SYSTEM TESTBED_MVCL (* Testbed Model/View/Control with Local Coupling *)
  (* Standard: 61499 ITA; Classification: Testbed *)
  (* Version 0.3, 2004-11-09, JHC, Rockwell Automation, Changed LOADL to LOADLE in CHAIN_MDL. *)
  (* Version 0.2, 2004-10-28, JHC, Rockwell Automation, Changed RING_FEED to CNVG_MDLL. *)
  (* Version 0.1, 2004-10-25, JHC, Rockwell Automation, Updated for new Load/Unload model. *)
  (* Version 0.0, 2004-09-22, JHC, Rockwell Automation *)
  DEVICE CONTROL : FRAME_DEVICE
    RESOURCE SORT : EMB_RES
      FBS
        SORT_PEG_SENSE : SUBL_2;
        RING_FEED_SENSE : SUBL_1;
        CTL : SORT_CTL;
        SORT_ACT : PUBL_1;
        LOST : E_PERMIT; (* RING_LOST event trigger *)
        RING_LOST : PUBL_0;
      END_FBS
      EVENT_CONNECTIONS
        START.COLD TO SORT_PEG_SENSE.INIT;
        SORT_PEG_SENSE.INITO TO RING_FEED_SENSE.INIT;
        RING_FEED_SENSE.INITO TO SORT_ACT.INIT;
        SORT_PEG_SENSE.IND TO CTL.REQ;
        CTL.CNF TO SORT_ACT.REQ;
        CTL.CNF TO LOST.EI;
        SORT_ACT.INITO TO RING_LOST.INIT;
        LOST.EO TO RING_LOST.REQ;
      END_CONNECTIONS
      DATA_CONNECTIONS
        RING_FEED_SENSE.RD_1 TO CTL.RING_PRESENT;
        CTL.SORT_SOLENOID TO SORT_ACT.SD_1;
        SORT_PEG_SENSE.RD_1 TO CTL.SORT_AREA_DETECT;
        SORT_PEG_SENSE.RD_2 TO CTL.METAL_PEG_DETECT;
        CTL.RING_LOST TO LOST.PERMIT;
      END_CONNECTIONS
    END_RESOURCE
    RESOURCE FEED : EMB_RES
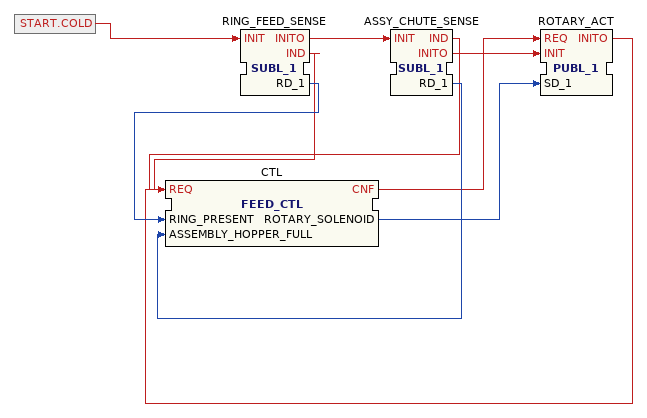
      FBS
        RING_FEED_SENSE : SUBL_1;
        ASSY_CHUTE_SENSE : SUBL_1;
        CTL : FEED_CTL;
        ROTARY_ACT : PUBL_1;
      END_FBS
      EVENT_CONNECTIONS
        START.COLD TO RING_FEED_SENSE.INIT;
        RING_FEED_SENSE.INITO TO ASSY_CHUTE_SENSE.INIT;
        ROTARY_ACT.INITO TO CTL.REQ;
        RING_FEED_SENSE.IND TO CTL.REQ;
        ASSY_CHUTE_SENSE.IND TO CTL.REQ;
        CTL.CNF TO ROTARY_ACT.REQ;
        ASSY_CHUTE_SENSE.INITO TO ROTARY_ACT.INIT;
      END_CONNECTIONS
      DATA_CONNECTIONS
        RING_FEED_SENSE.RD_1 TO CTL.RING_PRESENT;
        ASSY_CHUTE_SENSE.RD_1 TO CTL.ASSEMBLY_HOPPER_FULL;
        CTL.ROTARY_SOLENOID TO ROTARY_ACT.SD_1;
      END_CONNECTIONS
    END_RESOURCE
    RESOURCE INSPECT : EMB_RES
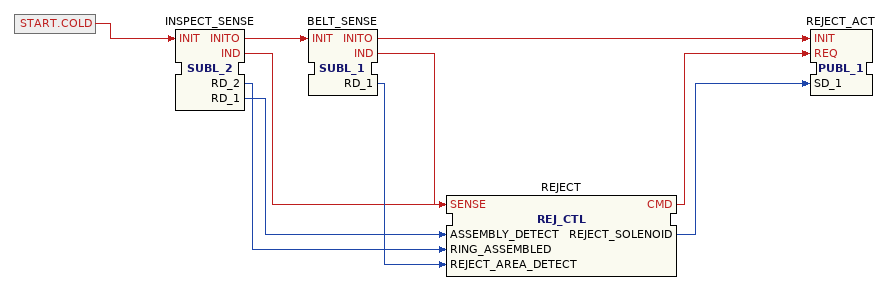
      FBS
        INSPECT_SENSE : SUBL_2;
        BELT_SENSE : SUBL_1;
        REJECT_ACT : PUBL_1;
        REJECT : REJ_CTL;
      END_FBS
      EVENT_CONNECTIONS
        START.COLD TO INSPECT_SENSE.INIT;
        INSPECT_SENSE.INITO TO BELT_SENSE.INIT;
        BELT_SENSE.INITO TO REJECT_ACT.INIT;
        INSPECT_SENSE.IND TO REJECT.SENSE;
        BELT_SENSE.IND TO REJECT.SENSE;
        REJECT.CMD TO REJECT_ACT.REQ;
      END_CONNECTIONS
      DATA_CONNECTIONS
        REJECT.REJECT_SOLENOID TO REJECT_ACT.SD_1;
        INSPECT_SENSE.RD_2 TO REJECT.RING_ASSEMBLED;
        INSPECT_SENSE.RD_1 TO REJECT.ASSEMBLY_DETECT;
        BELT_SENSE.RD_1 TO REJECT.REJECT_AREA_DETECT;
      END_CONNECTIONS
    END_RESOURCE
    RESOURCE CHAIN_SENSORS : PANEL_RESOURCE
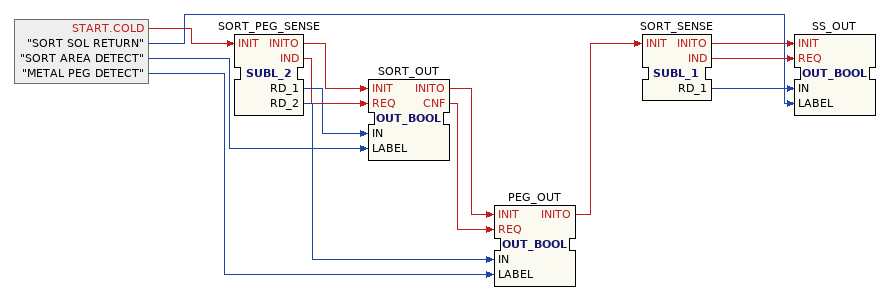
      FBS
        SORT_SENSE : SUBL_1;
        SS_OUT : OUT_BOOL;
        SORT_PEG_SENSE : SUBL_2;
        PEG_OUT : OUT_BOOL;
        SORT_OUT : OUT_BOOL;
      END_FBS
      EVENT_CONNECTIONS
        SORT_PEG_SENSE.INITO TO SORT_OUT.INIT;
        SORT_PEG_SENSE.IND TO SORT_OUT.REQ;
        SORT_OUT.INITO TO PEG_OUT.INIT;
        SORT_OUT.CNF TO PEG_OUT.REQ;
        START.COLD TO SORT_PEG_SENSE.INIT;
        PEG_OUT.INITO TO SORT_SENSE.INIT;
        SORT_SENSE.INITO TO SS_OUT.INIT;
        SORT_SENSE.IND TO SS_OUT.REQ;
      END_CONNECTIONS
      DATA_CONNECTIONS
        SORT_SENSE.RD_1 TO SS_OUT.IN;
        SORT_PEG_SENSE.RD_1 TO SORT_OUT.IN;
        SORT_PEG_SENSE.RD_2 TO PEG_OUT.IN;
        "SORT SOL RETURN" TO SS_OUT.LABEL;
        "SORT AREA DETECT" TO SORT_OUT.LABEL;
        "METAL PEG DETECT" TO PEG_OUT.LABEL;
      END_CONNECTIONS
    END_RESOURCE
    RESOURCE CHAIN_ACTUATORS : PANEL_RESOURCE
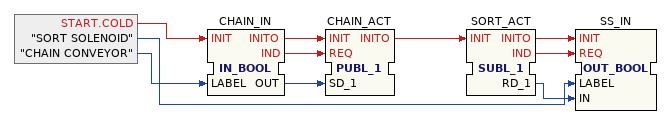
      FBS
        CHAIN_IN : IN_BOOL;
        CHAIN_ACT : PUBL_1;
        SS_IN : OUT_BOOL;
        SORT_ACT : SUBL_1;
      END_FBS
      EVENT_CONNECTIONS
        SORT_ACT.INITO TO SS_IN.INIT;
        SORT_ACT.IND TO SS_IN.REQ;
        START.COLD TO CHAIN_IN.INIT;
        CHAIN_IN.INITO TO CHAIN_ACT.INIT;
        CHAIN_ACT.INITO TO SORT_ACT.INIT;
        CHAIN_IN.IND TO CHAIN_ACT.REQ;
      END_CONNECTIONS
      DATA_CONNECTIONS
        "SORT SOLENOID" TO SS_IN.LABEL;
        "CHAIN CONVEYOR" TO CHAIN_IN.LABEL;
        SORT_ACT.RD_1 TO SS_IN.IN;
        CHAIN_IN.OUT TO CHAIN_ACT.SD_1;
      END_CONNECTIONS
    END_RESOURCE
    RESOURCE CHUTE_SENSORS : PANEL_RESOURCE
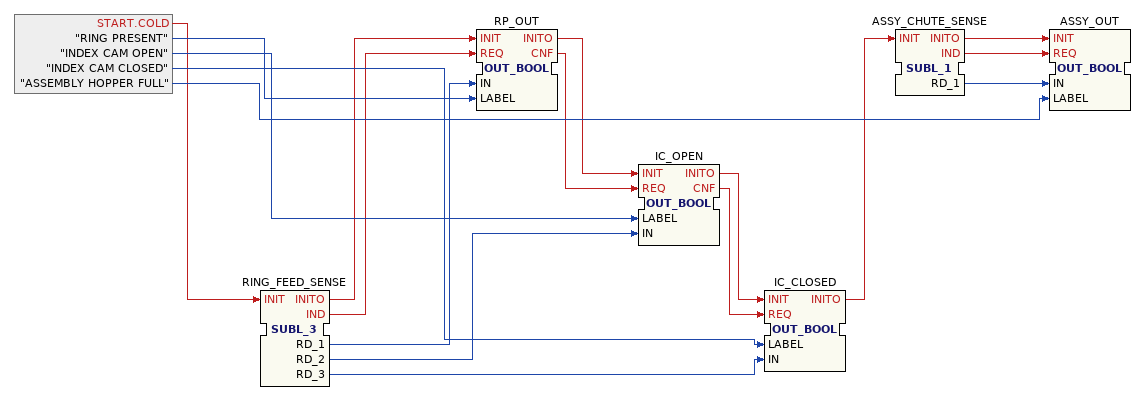
      FBS
        RING_FEED_SENSE : SUBL_3;
        RP_OUT : OUT_BOOL;
        IC_OPEN : OUT_BOOL;
        IC_CLOSED : OUT_BOOL;
        ASSY_CHUTE_SENSE : SUBL_1;
        ASSY_OUT : OUT_BOOL;
      END_FBS
      EVENT_CONNECTIONS
        START.COLD TO RING_FEED_SENSE.INIT;
        RING_FEED_SENSE.INITO TO RP_OUT.INIT;
        IC_OPEN.INITO TO IC_CLOSED.INIT;
        IC_CLOSED.INITO TO ASSY_CHUTE_SENSE.INIT;
        ASSY_CHUTE_SENSE.INITO TO ASSY_OUT.INIT;
        RING_FEED_SENSE.IND TO RP_OUT.REQ;
        IC_OPEN.CNF TO IC_CLOSED.REQ;
        ASSY_CHUTE_SENSE.IND TO ASSY_OUT.REQ;
        RP_OUT.INITO TO IC_OPEN.INIT;
        RP_OUT.CNF TO IC_OPEN.REQ;
      END_CONNECTIONS
      DATA_CONNECTIONS
        RING_FEED_SENSE.RD_1 TO RP_OUT.IN;
        "RING PRESENT" TO RP_OUT.LABEL;
        "INDEX CAM OPEN" TO IC_OPEN.LABEL;
        "INDEX CAM CLOSED" TO IC_CLOSED.LABEL;
        ASSY_CHUTE_SENSE.RD_1 TO ASSY_OUT.IN;
        "ASSEMBLY HOPPER FULL" TO ASSY_OUT.LABEL;
        RING_FEED_SENSE.RD_2 TO IC_OPEN.IN;
        RING_FEED_SENSE.RD_3 TO IC_CLOSED.IN;
      END_CONNECTIONS
    END_RESOURCE
    RESOURCE CHUTE_ACTUATORS : PANEL_RESOURCE
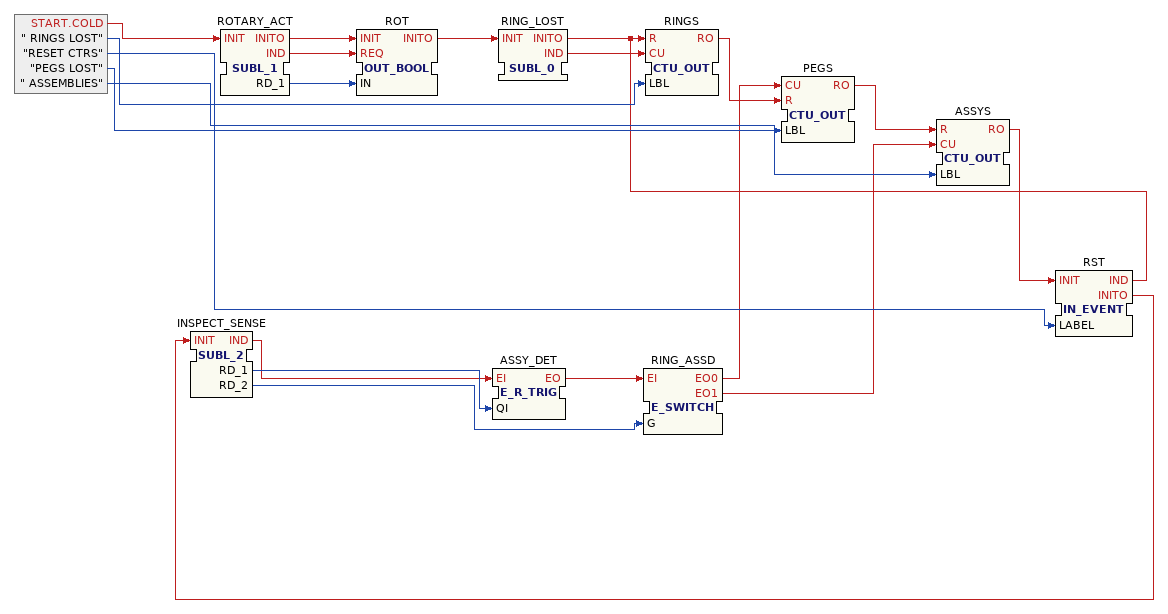
      FBS
        ROT : OUT_BOOL;
        ROTARY_ACT : SUBL_1;
        RING_LOST : SUBL_0;
        RINGS : CTU_OUT;
        RST : IN_EVENT;
        PEGS : CTU_OUT;
        ASSYS : CTU_OUT;
        ASSY_DET : E_R_TRIG; (* QI = ASSEMBLY_DETECT *)
        RING_ASSD : E_SWITCH; (* G = RING_ASSEMBLED *)
        INSPECT_SENSE : SUBL_2;
      END_FBS
      EVENT_CONNECTIONS
        START.COLD TO ROTARY_ACT.INIT;
        ROTARY_ACT.INITO TO ROT.INIT;
        ROTARY_ACT.IND TO ROT.REQ;
        ROT.INITO TO RING_LOST.INIT;
        RING_LOST.INITO TO RINGS.R;
        RING_LOST.IND TO RINGS.CU;
        RST.IND TO RINGS.R;
        ASSYS.RO TO RST.INIT;
        ASSY_DET.EO TO RING_ASSD.EI;
        INSPECT_SENSE.IND TO ASSY_DET.EI;
        RING_ASSD.EO0 TO PEGS.CU;
        RINGS.RO TO PEGS.R;
        PEGS.RO TO ASSYS.R;
        RING_ASSD.EO1 TO ASSYS.CU;
        RST.INITO TO INSPECT_SENSE.INIT;
      END_CONNECTIONS
      DATA_CONNECTIONS
        " RINGS LOST" TO RINGS.LBL;
        "RESET CTRS" TO RST.LABEL;
        "PEGS LOST" TO PEGS.LBL;
        " ASSEMBLIES" TO ASSYS.LBL;
        INSPECT_SENSE.RD_1 TO ASSY_DET.QI;
        INSPECT_SENSE.RD_2 TO RING_ASSD.G;
        ROTARY_ACT.RD_1 TO ROT.IN;
      END_CONNECTIONS
    END_RESOURCE
    RESOURCE BELT_SENSORS : PANEL_RESOURCE
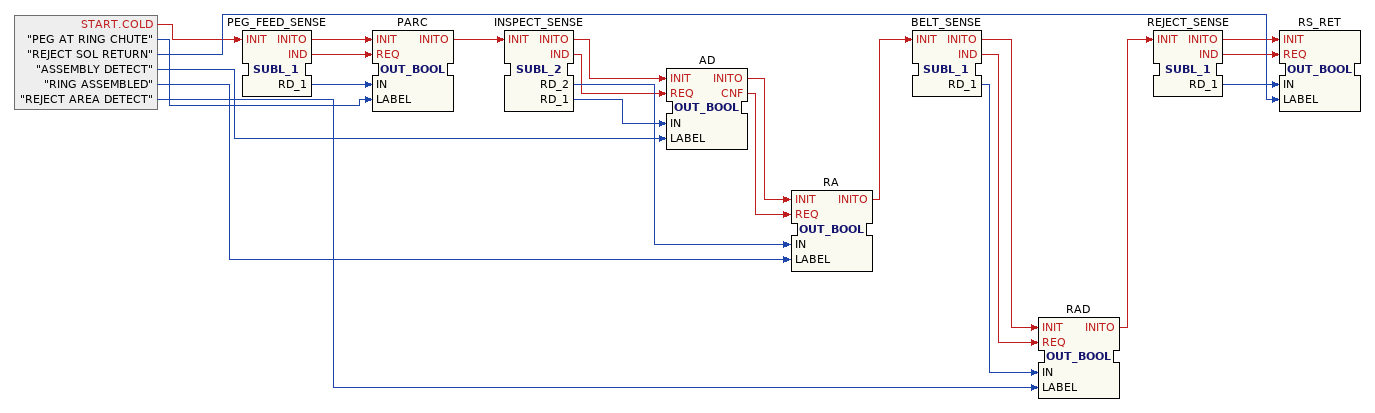
      FBS
        PEG_FEED_SENSE : SUBL_1;
        PARC : OUT_BOOL;
        INSPECT_SENSE : SUBL_2;
        AD : OUT_BOOL;
        RA : OUT_BOOL;
        BELT_SENSE : SUBL_1;
        RAD : OUT_BOOL;
        REJECT_SENSE : SUBL_1;
        RS_RET : OUT_BOOL;
      END_FBS
      EVENT_CONNECTIONS
        START.COLD TO PEG_FEED_SENSE.INIT;
        PEG_FEED_SENSE.INITO TO PARC.INIT;
        PARC.INITO TO INSPECT_SENSE.INIT;
        INSPECT_SENSE.INITO TO AD.INIT;
        AD.INITO TO RA.INIT;
        RA.INITO TO BELT_SENSE.INIT;
        BELT_SENSE.INITO TO RAD.INIT;
        RAD.INITO TO REJECT_SENSE.INIT;
        REJECT_SENSE.INITO TO RS_RET.INIT;
        PEG_FEED_SENSE.IND TO PARC.REQ;
        INSPECT_SENSE.IND TO AD.REQ;
        AD.CNF TO RA.REQ;
        BELT_SENSE.IND TO RAD.REQ;
        REJECT_SENSE.IND TO RS_RET.REQ;
      END_CONNECTIONS
      DATA_CONNECTIONS
        PEG_FEED_SENSE.RD_1 TO PARC.IN;
        "PEG AT RING CHUTE" TO PARC.LABEL;
        REJECT_SENSE.RD_1 TO RS_RET.IN;
        "REJECT SOL RETURN" TO RS_RET.LABEL;
        INSPECT_SENSE.RD_2 TO RA.IN;
        INSPECT_SENSE.RD_1 TO AD.IN;
        "ASSEMBLY DETECT" TO AD.LABEL;
        "RING ASSEMBLED" TO RA.LABEL;
        BELT_SENSE.RD_1 TO RAD.IN;
        "REJECT AREA DETECT" TO RAD.LABEL;
      END_CONNECTIONS
    END_RESOURCE
    RESOURCE BELT_ACTUATORS : PANEL_RESOURCE
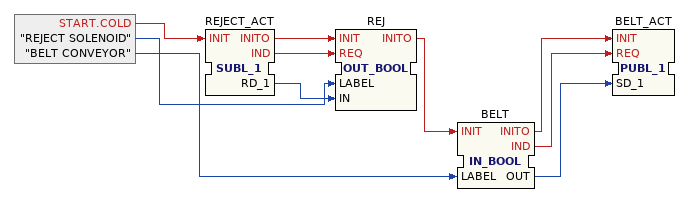
      FBS
        REJ : OUT_BOOL;
        REJECT_ACT : SUBL_1;
        BELT : IN_BOOL;
        BELT_ACT : PUBL_1;
      END_FBS
      EVENT_CONNECTIONS
        BELT.INITO TO BELT_ACT.INIT;
        BELT.IND TO BELT_ACT.REQ;
        START.COLD TO REJECT_ACT.INIT;
        REJECT_ACT.INITO TO REJ.INIT;
        REJECT_ACT.IND TO REJ.REQ;
        REJ.INITO TO BELT.INIT;
      END_CONNECTIONS
      DATA_CONNECTIONS
        "REJECT SOLENOID" TO REJ.LABEL;
        BELT.OUT TO BELT_ACT.SD_1;
        "BELT CONVEYOR" TO BELT.LABEL;
        REJECT_ACT.RD_1 TO REJ.IN;
      END_CONNECTIONS
    END_RESOURCE
  END_DEVICE
  DEVICE MODEL : FRAME_DEVICE
    RESOURCE CLOCK : EMB_RES
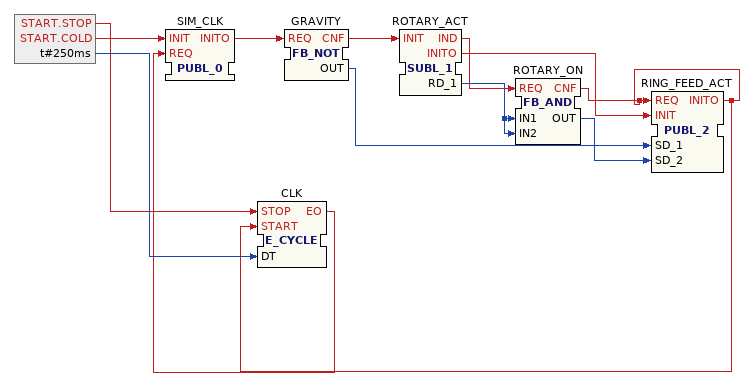
      FBS
        CLK : E_CYCLE;
        SIM_CLK : PUBL_0;
        GRAVITY : FB_NOT;
        ROTARY_ACT : SUBL_1;
        ROTARY_ON : FB_AND;
        RING_FEED_ACT : PUBL_2;
      END_FBS
      EVENT_CONNECTIONS
        START.STOP TO CLK.STOP;
        START.COLD TO SIM_CLK.INIT;
        CLK.EO TO SIM_CLK.REQ;
        SIM_CLK.INITO TO GRAVITY.REQ;
        GRAVITY.CNF TO ROTARY_ACT.INIT;
        ROTARY_ACT.IND TO ROTARY_ON.REQ;
        ROTARY_ON.CNF TO RING_FEED_ACT.REQ;
        ROTARY_ACT.INITO TO RING_FEED_ACT.INIT;
        RING_FEED_ACT.INITO TO RING_FEED_ACT.REQ;
        RING_FEED_ACT.INITO TO CLK.START;
      END_CONNECTIONS
      DATA_CONNECTIONS
        t#250ms TO CLK.DT;
        GRAVITY.OUT TO RING_FEED_ACT.SD_1;
        ROTARY_ACT.RD_1 TO ROTARY_ON.IN1;
        ROTARY_ACT.RD_1 TO ROTARY_ON.IN2;
        ROTARY_ON.OUT TO RING_FEED_ACT.SD_2;
      END_CONNECTIONS
    END_RESOURCE
    RESOURCE CHAIN_MDL : EMB_RES
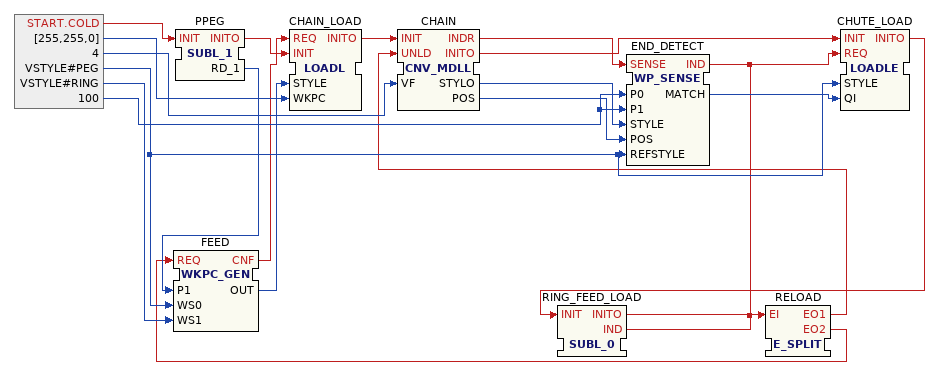
      FBS
        PPEG : SUBL_1;
        FEED : WKPC_GEN;
        CHAIN : CNV_MDLL;
        RING_FEED_LOAD : SUBL_0;
        END_DETECT : WP_SENSE;
        CHAIN_LOAD : LOADL;
        RELOAD : E_SPLIT;
        CHUTE_LOAD : LOADLE;
      END_FBS
      EVENT_CONNECTIONS
        FEED.CNF TO CHAIN_LOAD.REQ;
        START.COLD TO PPEG.INIT;
        PPEG.INITO TO CHAIN_LOAD.INIT;
        CHAIN_LOAD.INITO TO CHAIN.INIT;
        RELOAD.EO1 TO CHAIN.UNLD;
        RELOAD.EO2 TO FEED.REQ;
        RING_FEED_LOAD.INITO TO RELOAD.EI;
        RING_FEED_LOAD.IND TO RELOAD.EI;
        CHAIN.INDR TO END_DETECT.SENSE;
        CHAIN.INITO TO CHUTE_LOAD.INIT;
        CHUTE_LOAD.INITO TO RING_FEED_LOAD.INIT;
        END_DETECT.IND TO CHUTE_LOAD.REQ;
        END_DETECT.IND TO RELOAD.EI;
      END_CONNECTIONS
      DATA_CONNECTIONS
        FEED.OUT TO CHAIN_LOAD.STYLE;
        [255,255,0] TO CHAIN_LOAD.WKPC;
        4 TO CHAIN.VF; (* 16% per sec =100% per 6.25 sec *)
        PPEG.RD_1 TO FEED.P1;
        VSTYLE#PEG TO FEED.WS0;
        VSTYLE#RING TO FEED.WS1;
        100 TO END_DETECT.P0;
        100 TO END_DETECT.P1;
        CHAIN.STYLO TO END_DETECT.STYLE;
        CHAIN.POS TO END_DETECT.POS;
        VSTYLE#PEG TO END_DETECT.REFSTYLE;
        VSTYLE#PEG TO CHUTE_LOAD.STYLE;
        END_DETECT.MATCH TO CHUTE_LOAD.QI;
      END_CONNECTIONS
    END_RESOURCE
    RESOURCE SORT_MDL : EMB_RES
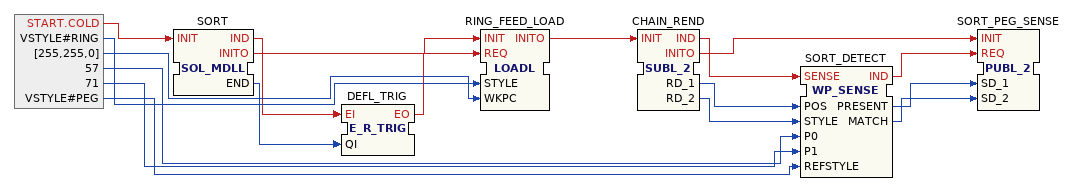
      FBS
        SORT : SOL_MDLL;
        DEFL_TRIG : E_R_TRIG;
        RING_FEED_LOAD : LOADL;
        CHAIN_REND : SUBL_2;
        SORT_DETECT : WP_SENSE;
        SORT_PEG_SENSE : PUBL_2;
      END_FBS
      EVENT_CONNECTIONS
        START.COLD TO SORT.INIT;
        SORT.IND TO DEFL_TRIG.EI;
        SORT.INITO TO RING_FEED_LOAD.INIT;
        DEFL_TRIG.EO TO RING_FEED_LOAD.REQ;
        RING_FEED_LOAD.INITO TO CHAIN_REND.INIT;
        CHAIN_REND.IND TO SORT_DETECT.SENSE;
        CHAIN_REND.INITO TO SORT_PEG_SENSE.INIT;
        SORT_DETECT.IND TO SORT_PEG_SENSE.REQ;
      END_CONNECTIONS
      DATA_CONNECTIONS
        VSTYLE#RING TO RING_FEED_LOAD.STYLE;
        [255,255,0] TO RING_FEED_LOAD.WKPC;
        SORT.END TO DEFL_TRIG.QI;
        CHAIN_REND.RD_1 TO SORT_DETECT.POS;
        CHAIN_REND.RD_2 TO SORT_DETECT.STYLE;
        57 TO SORT_DETECT.P0;
        71 TO SORT_DETECT.P1;
        VSTYLE#PEG TO SORT_DETECT.REFSTYLE;
        SORT_DETECT.PRESENT TO SORT_PEG_SENSE.SD_1;
        SORT_DETECT.MATCH TO SORT_PEG_SENSE.SD_2;
      END_CONNECTIONS
    END_RESOURCE
    RESOURCE PEG_CHUTE : EMB_RES
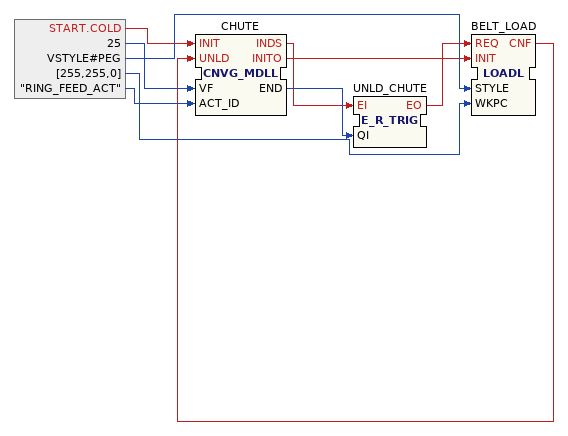
      FBS
        CHUTE : CNVG_MDLL;
        UNLD_CHUTE : E_R_TRIG;
        BELT_LOAD : LOADL;
      END_FBS
      EVENT_CONNECTIONS
        CHUTE.INDS TO UNLD_CHUTE.EI;
        START.COLD TO CHUTE.INIT;
        UNLD_CHUTE.EO TO BELT_LOAD.REQ;
        BELT_LOAD.CNF TO CHUTE.UNLD;
        CHUTE.INITO TO BELT_LOAD.INIT;
      END_CONNECTIONS
      DATA_CONNECTIONS
        25 TO CHUTE.VF; (* 2 sec FS *)
        CHUTE.END TO UNLD_CHUTE.QI;
        VSTYLE#PEG TO BELT_LOAD.STYLE;
        [255,255,0] TO BELT_LOAD.WKPC;
        "RING_FEED_ACT" TO CHUTE.ACT_ID;
      END_CONNECTIONS
    END_RESOURCE
    RESOURCE RING_CHUTES : EMB_RES
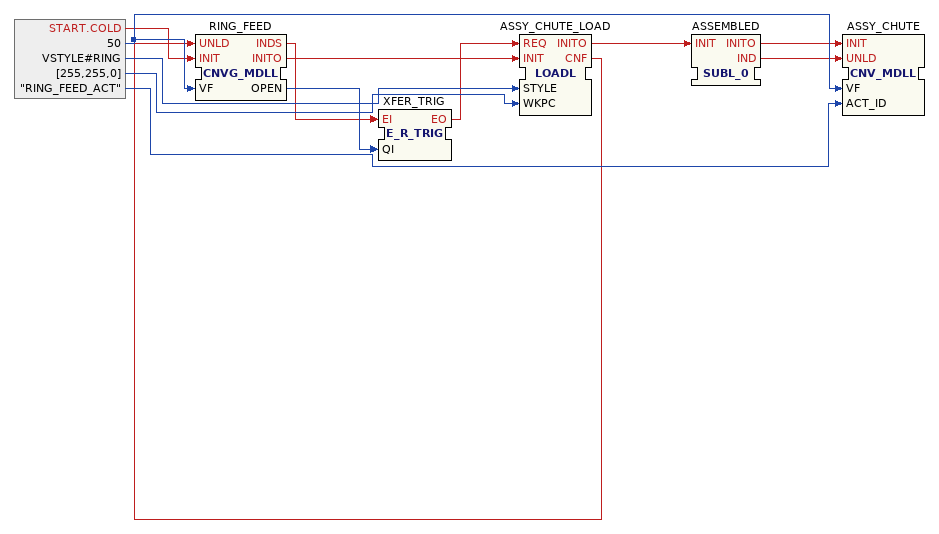
      FBS
        RING_FEED : CNVG_MDLL;
        ASSY_CHUTE : CNV_MDLL;
        XFER_TRIG : E_R_TRIG;
        ASSY_CHUTE_LOAD : LOADL;
        ASSEMBLED : SUBL_0;
      END_FBS
      EVENT_CONNECTIONS
        XFER_TRIG.EO TO ASSY_CHUTE_LOAD.REQ;
        ASSY_CHUTE_LOAD.INITO TO ASSEMBLED.INIT;
        RING_FEED.INDS TO XFER_TRIG.EI;
        ASSY_CHUTE_LOAD.CNF TO RING_FEED.UNLD;
        START.COLD TO RING_FEED.INIT;
        RING_FEED.INITO TO ASSY_CHUTE_LOAD.INIT;
        ASSEMBLED.INITO TO ASSY_CHUTE.INIT;
        ASSEMBLED.IND TO ASSY_CHUTE.UNLD;
      END_CONNECTIONS
      DATA_CONNECTIONS
        50 TO ASSY_CHUTE.VF; (* 500 ms full scale *)
        50 TO RING_FEED.VF; (* 500ms Full Scale *)
        VSTYLE#RING TO ASSY_CHUTE_LOAD.STYLE;
        [255,255,0] TO ASSY_CHUTE_LOAD.WKPC;
        RING_FEED.OPEN TO XFER_TRIG.QI;
        "RING_FEED_ACT" TO ASSY_CHUTE.ACT_ID;
      END_CONNECTIONS
    END_RESOURCE
    RESOURCE BELT_MDL : EMB_RES
      FBS
        BELT : CNV_MDLL;
        REJECT : SOL_MDLL;
        END_TRIG : E_R_TRIG;
        END_DLY : CL_DELAY;
      END_FBS
      EVENT_CONNECTIONS
        END_TRIG.EO TO END_DLY.START;
        END_DLY.EO TO BELT.UNLD;
        END_DLY.INITO TO REJECT.INIT;
        BELT.INDS TO END_TRIG.EI;
        BELT.INITO TO END_DLY.INIT;
        START.COLD TO BELT.INIT;
      END_CONNECTIONS
      DATA_CONNECTIONS
        5 TO BELT.VF; (* 20% per sec = 5 sec Full Scale *)
        BELT.END TO END_TRIG.QI;
        3 TO END_DLY.N;
      END_CONNECTIONS
    END_RESOURCE
    RESOURCE ASSY_MDL : EMB_RES (* Model for Peg/Ring Assembly *)
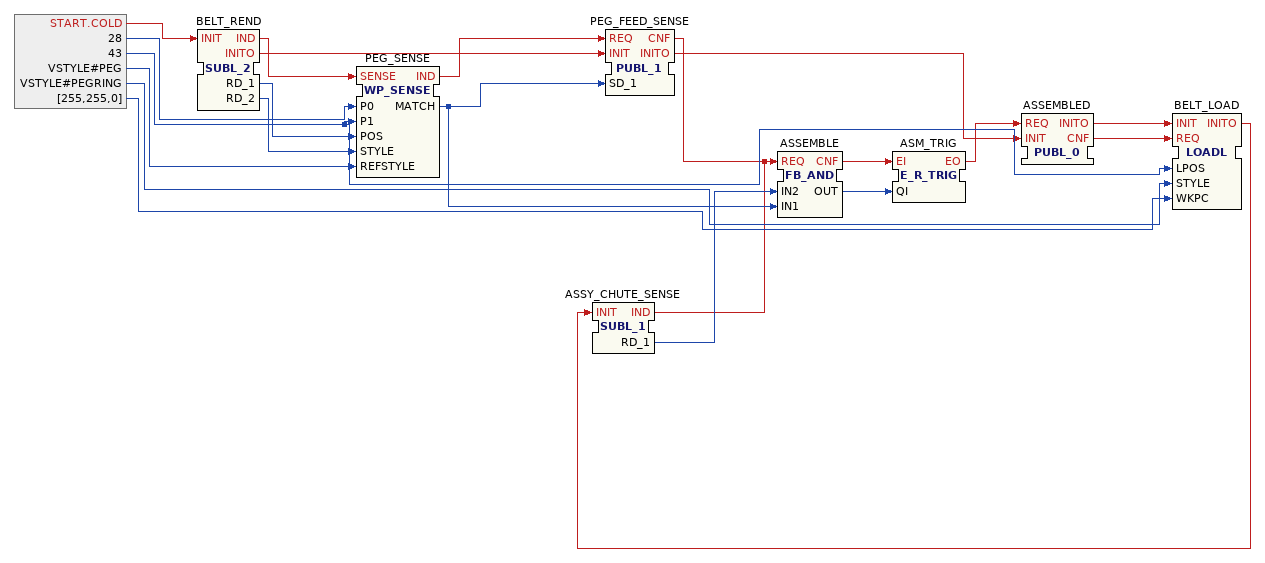
      FBS
        PEG_SENSE : WP_SENSE;
        PEG_FEED_SENSE : PUBL_1;
        ASSY_CHUTE_SENSE : SUBL_1;
        ASSEMBLE : FB_AND;
        ASM_TRIG : E_R_TRIG;
        BELT_REND : SUBL_2;
        ASSEMBLED : PUBL_0;
        BELT_LOAD : LOADL;
      END_FBS
      EVENT_CONNECTIONS
        PEG_SENSE.IND TO PEG_FEED_SENSE.REQ;
        PEG_FEED_SENSE.CNF TO ASSEMBLE.REQ;
        ASSEMBLE.CNF TO ASM_TRIG.EI;
        START.COLD TO BELT_REND.INIT;
        BELT_REND.IND TO PEG_SENSE.SENSE;
        BELT_REND.INITO TO PEG_FEED_SENSE.INIT;
        ASM_TRIG.EO TO ASSEMBLED.REQ;
        PEG_FEED_SENSE.INITO TO ASSEMBLED.INIT;
        ASSY_CHUTE_SENSE.IND TO ASSEMBLE.REQ;
        ASSEMBLED.INITO TO BELT_LOAD.INIT;
        ASSEMBLED.CNF TO BELT_LOAD.REQ;
        BELT_LOAD.INITO TO ASSY_CHUTE_SENSE.INIT;
      END_CONNECTIONS
      DATA_CONNECTIONS
        28 TO PEG_SENSE.P0; (* =2/7 *)
        43 TO PEG_SENSE.P1; (* =3/7 *)
        ASSEMBLE.OUT TO ASM_TRIG.QI;
        BELT_REND.RD_1 TO PEG_SENSE.POS;
        BELT_REND.RD_2 TO PEG_SENSE.STYLE;
        PEG_SENSE.MATCH TO PEG_FEED_SENSE.SD_1;
        ASSY_CHUTE_SENSE.RD_1 TO ASSEMBLE.IN2;
        PEG_SENSE.MATCH TO ASSEMBLE.IN1;
        VSTYLE#PEG TO PEG_SENSE.REFSTYLE;
        43 TO BELT_LOAD.LPOS;
        VSTYLE#PEGRING TO BELT_LOAD.STYLE;
        [255,255,0] TO BELT_LOAD.WKPC;
      END_CONNECTIONS
    END_RESOURCE
    RESOURCE INSP_MDL : EMB_RES (* Inspection Model *)
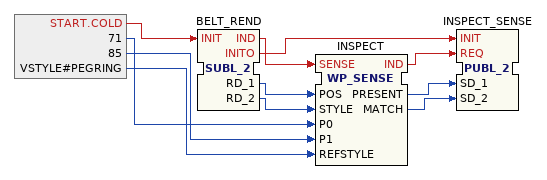
      FBS
        BELT_REND : SUBL_2;
        INSPECT : WP_SENSE;
        INSPECT_SENSE : PUBL_2;
      END_FBS
      EVENT_CONNECTIONS
        START.COLD TO BELT_REND.INIT;
        BELT_REND.IND TO INSPECT.SENSE;
        BELT_REND.INITO TO INSPECT_SENSE.INIT;
        INSPECT.IND TO INSPECT_SENSE.REQ;
      END_CONNECTIONS
      DATA_CONNECTIONS
        BELT_REND.RD_1 TO INSPECT.POS;
        BELT_REND.RD_2 TO INSPECT.STYLE;
        71 TO INSPECT.P0; (* =5/7 *)
        85 TO INSPECT.P1; (* =6/7 *)
        INSPECT.PRESENT TO INSPECT_SENSE.SD_1;
        INSPECT.MATCH TO INSPECT_SENSE.SD_2;
        VSTYLE#PEGRING TO INSPECT.REFSTYLE;
      END_CONNECTIONS
    END_RESOURCE
    RESOURCE CHAIN : VIEW_PANEL
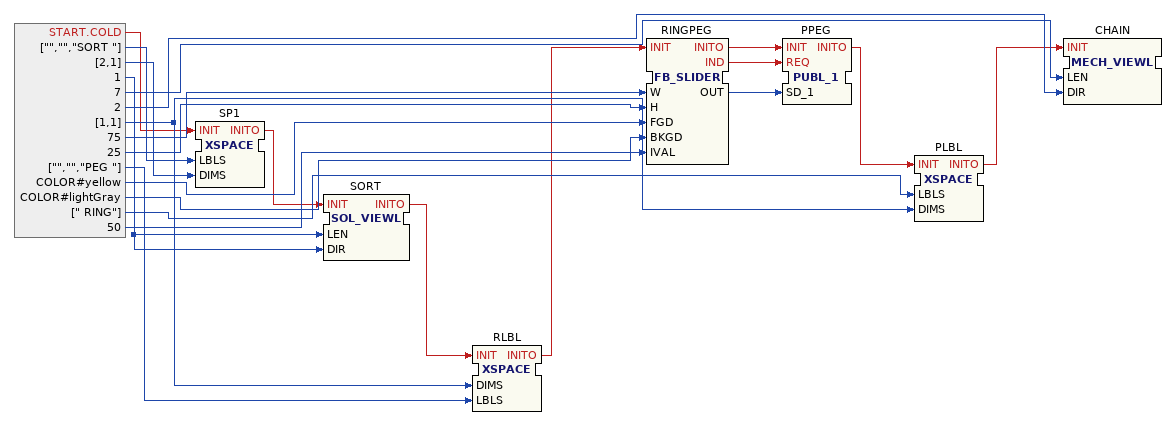
      FBS
        SP1 : XSPACE;
        SORT : SOL_VIEWL; (* Sort Solenoid *)
        RLBL : XSPACE;
        CHAIN : MECH_VIEWL; (* First Chain Segment *)
        RINGPEG : FB_SLIDER;
        PLBL : XSPACE;
        PPEG : PUBL_1; (* Peg probability (0-100) *)
      END_FBS
      EVENT_CONNECTIONS
        START.COLD TO SP1.INIT;
        SP1.INITO TO SORT.INIT;
        SORT.INITO TO RLBL.INIT;
        RLBL.INITO TO RINGPEG.INIT;
        RINGPEG.INITO TO PPEG.INIT;
        PPEG.INITO TO PLBL.INIT;
        RINGPEG.IND TO PPEG.REQ;
        PLBL.INITO TO CHAIN.INIT;
      END_CONNECTIONS
      DATA_CONNECTIONS
        ["","","SORT "] TO SP1.LBLS;
        [2,1] TO SP1.DIMS;
        1 TO SORT.LEN;
        1 TO SORT.DIR;
        7 TO CHAIN.LEN;
        2 TO CHAIN.DIR;
        [1,1] TO RLBL.DIMS;
        75 TO RINGPEG.W;
        25 TO RINGPEG.H;
        ["","","PEG "] TO RLBL.LBLS;
        COLOR#yellow TO RINGPEG.FGD;
        COLOR#lightGray TO RINGPEG.BKGD;
        [" RING"] TO PLBL.LBLS;
        [1,1] TO PLBL.DIMS;
        RINGPEG.OUT TO PPEG.SD_1;
        50 TO RINGPEG.IVAL;
      END_CONNECTIONS
    END_RESOURCE
    RESOURCE CHUTES : VIEW_PANEL
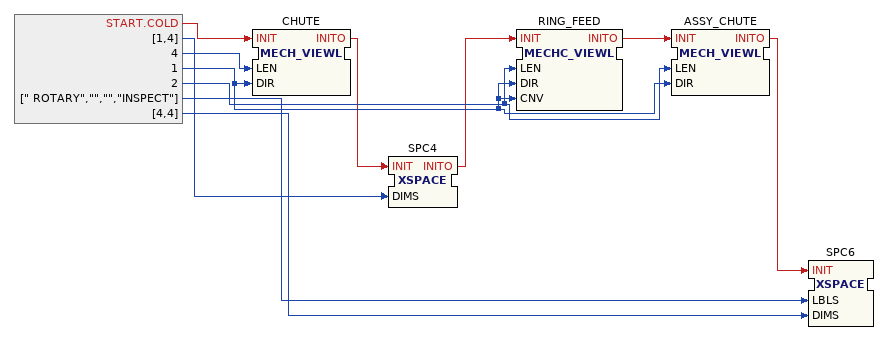
      FBS
        CHUTE : MECH_VIEWL; (* Peg Chute *)
        SPC4 : XSPACE; (* Ring Feed Chute *)
        RING_FEED : MECHC_VIEWL; (* Ring Feed Chute *)
        ASSY_CHUTE : MECH_VIEWL; (* Assembly Chute *)
        SPC6 : XSPACE;
      END_FBS
      EVENT_CONNECTIONS
        START.COLD TO CHUTE.INIT;
        CHUTE.INITO TO SPC4.INIT;
        SPC4.INITO TO RING_FEED.INIT;
        RING_FEED.INITO TO ASSY_CHUTE.INIT;
        ASSY_CHUTE.INITO TO SPC6.INIT;
      END_CONNECTIONS
      DATA_CONNECTIONS
        [1,4] TO SPC4.DIMS;
        4 TO CHUTE.LEN;
        1 TO CHUTE.DIR;
        2 TO RING_FEED.LEN;
        1 TO RING_FEED.DIR;
        2 TO ASSY_CHUTE.LEN;
        1 TO ASSY_CHUTE.DIR;
        [" ROTARY","","","INSPECT"] TO SPC6.LBLS;
        [4,4] TO SPC6.DIMS;
        1 TO RING_FEED.CNV;
      END_CONNECTIONS
    END_RESOURCE
    RESOURCE BELT : VIEW_PANEL
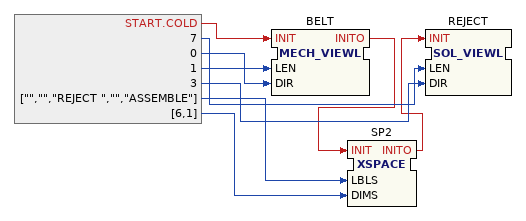
      FBS
        BELT : MECH_VIEWL;
        SP2 : XSPACE;
        REJECT : SOL_VIEWL;
      END_FBS
      EVENT_CONNECTIONS
        START.COLD TO BELT.INIT;
        SP2.INITO TO REJECT.INIT;
        BELT.INITO TO SP2.INIT;
      END_CONNECTIONS
      DATA_CONNECTIONS
        7 TO BELT.LEN;
        0 TO BELT.DIR;
        1 TO REJECT.LEN;
        3 TO REJECT.DIR;
        ["","","REJECT ","","ASSEMBLE"] TO SP2.LBLS;
        [6,1] TO SP2.DIMS;
      END_CONNECTIONS
    END_RESOURCE
    DATA_CONNECTIONS
      40 TO CHUTES.DIA;
      [7,4] TO CHUTES.SIZE;
      1 TO CHUTES.VERTICAL;
      40 TO BELT.DIA;
      [7,2] TO BELT.SIZE;
      0 TO CHAIN.TRACE;
      40 TO CHAIN.DIA;
      [7,2] TO CHAIN.SIZE;
    END_CONNECTIONS
  END_DEVICE
  DATA_CONNECTIONS (* parameter values *)
    [100,100,350,360] TO CONTROL.BOUNDS;
    [0,2] TO CONTROL.GRID;
    [450,100,290,360] TO MODEL.BOUNDS;
  END_CONNECTIONS
END_SYSTEM
